{attribute 'linkalways'} 
{attribute 'no_explicit_call' := 'This FB is a CLASS and must be accessed using methods or properties'}
{attribute 'enable_dynamic_creation'}
FUNCTION_BLOCK _DT EXTENDS DatatypeBase
VAR
	localData : DT;
	activeData : REFERENCE TO DT REF= localData;
END_VAR

PROPERTY PUBLIC Address : PVOID
GET
Address := ADR(activeData);
END_GET
END_PROPERTY

METHOD PUBLIC ClearReference
VAR_INPUT
END_VAR
activeData REF= localData;
END_METHOD

METHOD PUBLIC Clone : I_Datatype
VAR
    pClone : POINTER TO _DT;
END_VAR
pClone := __NEW(_DT(InitialValue := Value));
Clone := pClone^;
END_METHOD

METHOD FB_init : BOOL
VAR_INPUT
	bInitRetains : BOOL; // if TRUE, the retain variables are initialized (warm start / cold start)
	bInCopyCode : BOOL;  // if TRUE, the instance afterwards gets moved WORDo the copy code (online change)
	InitialValue : DT;
END_VAR
localData := InitialValue;
END_METHOD

METHOD PUBLIC MakeReferenceTo
VAR_INPUT
	ReferenceTarget : REFERENCE TO DT;
END_VAR
activeData REF= ReferenceTarget;
END_METHOD

METHOD PUBLIC SerializeWith
VAR_INPUT
	Serializer : I_Serializer;
END_VAR
Serializer.AddDateTime(activeData);
END_METHOD

PROPERTY PUBLIC Size : UDINT
GET
Size := SIZEOF(activeData);
END_GET
END_PROPERTY

METHOD TryDeserializeFrom : BOOL
VAR_INPUT
	Deserializer : I_Deserializer;
	Feedback : I_DeserializerFeedback;
END_VAR
TryDeserializeFrom := Deserializer.TryGetDateTime(activeData, Feedback);
END_METHOD

METHOD TryMakeReferenceTo : BOOL
VAR_INPUT
	Target : I_Datatype;
END_VAR
VAR
	pTargetData : POINTER TO DT;
END_VAR
IF NOT (Target.TypeName = TypeName) THEN
	RETURN;
END_IF

pTargetData := Target.Address;
activeData REF= pTargetData^;
TryMakeReferenceTo := TRUE;
END_METHOD

PROPERTY PUBLIC TypeName : T_MAXSTRING
GET
TypeName := 'DT';
END_GET
END_PROPERTY

PROPERTY PUBLIC Value : REFERENCE TO DT
GET
Value REF= activeData;
END_GET
END_PROPERTY

END_FUNCTION_BLOCK

(* stored: Version 1.1.0.1, ProductVersion 3.1.4024.12
   POU _DT: Id {fdfba514-5215-4b6c-a89a-973bdf10424c}, SpecialFunc None
   Folder Constructor: Id {b529c6b5-f3d7-4b92-9088-502ba7742fdd}
   Property Address: Id {5fa3e70f-47c5-4595-8d3e-4d1ca9668322}
   Get Get: Id {33b3fc2d-f3d2-4974-9222-edff81ccc6a0}
   Method ClearReference: Id {d20d8541-56de-4423-a36a-ca666cb1ff0f}
   Method Clone: Id {8d70687f-a9ac-4f50-af11-5539462c6a48}
   Method FB_init: Id {13537de6-70c4-475d-9122-2b33d4a5102b}
   Method MakeReferenceTo: Id {d91c301b-7fce-4e77-bd35-5ba215b1fad1}
   Method SerializeWith: Id {c77b2660-3a86-4f73-9d15-33ca60324fc4}
   Property Size: Id {17e7b6bd-6155-48a5-aa39-7195cbea4706}
   Get Get: Id {c6e0e203-efc2-457f-b016-ed463715c430}
   Method TryDeserializeFrom: Id {efcab989-b40b-4b1c-a574-60770556a9f4}
   Method TryMakeReferenceTo: Id {dabf4821-6b5f-4f8e-be0e-de26466bae86}
   Property TypeName: Id {1e365a3c-30cc-40e6-a6a7-db03c568f3e5}
   Get Get: Id {072a4dd1-aab7-4491-9a57-5d744dbd9605}
   Property Value: Id {994236d9-26f2-48e9-afc4-2298f7c33a37}
   Get Get: Id {dc2b5892-6a17-4f11-8a48-929cb26d660e} *)
